TYPE ST_OutputData_KL320x :
STRUCT
	usiControl			: USINT;				//Output Control from KL320x
	iDataOut			: INT;					//Output Data from KL320x
END_STRUCT
END_TYPE

(* stored: Version 1.1.0.1, ProductVersion 3.1.4024.6
   DUT ST_OutputData_KL320x: Id {973468c6-91b2-452f-b951-58f688f41112} *)
